Staubli VAL3: iRack1.pgx

public program iRack1(num& nNum[] (dimensions=1))
begin
  nNum=dioGet(iRack1)
end
